TYPE TcoTransferSystem_Control EXTENDS TcoCore.TcoStruct:
STRUCT

	
		
END_STRUCT
END_TYPE

(* stored: Version 1.1.0.1
   DUT TcoTransferSystem_Control: Id {8505063f-c790-4b12-9972-c262c881f17d} *)
